PROGRAM DemoProgram
VAR
	{attribute 'OPC.UA.DA' := '1'}
    //{attribute 'OPC.UA.DA.StructuredType' := '1'}
//	Events:EventsFB;
	
	fbProgramBase :FB_PrgmBasic;
	//EventParameters:EventParam_Typ;	
	flowid:DINT;
	testevent:BOOL;
	refEvent :REFERENCE TO EventHelper;
END_VAR


//EventParameters.par2:=2;
IF testevent THEN
	fbProgramBase.EventParameters.Par1:=1;
//	fbProgramBase.mEventThrow(ev_PLC_ILLEGAL_MSG,ADR(flowid),ADR(fbProgramBase.EventParameters));
	fbProgramBase.mEventThrow(ev_PLC_ILLEGAL_MSG,ADR(fbProgramBase.EventHeader),ADR(fbProgramBase.EventParameters));
	
	fbProgramBase.EventParameters.Par1:=3;
//	fbProgramBase.mEventThrow(ev_PLC_INTERNAL_TIMEOUT,ADR(flowid),ADR(fbProgramBase.EventParameters));
	fbProgramBase.mEventThrow(ev_PLC_INTERNAL_TIMEOUT,ADR(fbProgramBase.EventHeader),ADR(fbProgramBase.EventParameters));

		fbProgramBase.EventParameters.Par1:=5;
//	fbProgramBase.mEventThrow(ev_PLC_ILLEGAL_MSG,ADR(flowid),ADR(fbProgramBase.EventParameters));
	fbProgramBase.mEventThrow(ev_PLC_ILLEGAL_MSG,ADR(fbProgramBase.EventHeader),ADR(fbProgramBase.EventParameters));
	
		fbProgramBase.EventParameters.Par1:=3;
//	fbProgramBase.mEventThrow(ev_PLC_INTERNAL_TIMEOUT,ADR(flowid),ADR(fbProgramBase.EventParameters));
	fbProgramBase.mEventThrow(ev_PLC_INTERNAL_TIMEOUT,ADR(fbProgramBase.EventHeader),ADR(fbProgramBase.EventParameters));
	testevent:=FALSE;
END_IF


fbProgramBase();

END_PROGRAM

(* stored: Version 1.1.0.1, ProductVersion 3.1.4024.3
   POU DemoProgram: Id {2cb81fdf-e547-0e79-0a99-172c7a9c122b}, SpecialFunc None *)
